FUNCTION_BLOCK SifbManagementControls
  (* Standard: 61499-2 *)
  (* Version 0.1, 2019-00-29, hpea485, UOA *)
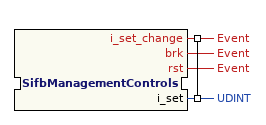
  EVENT_OUTPUT
    i_set_change WITH i_set;
    brk;
    rst;
  END_EVENT
  VAR_OUTPUT
    i_set : UDINT;
  END_VAR
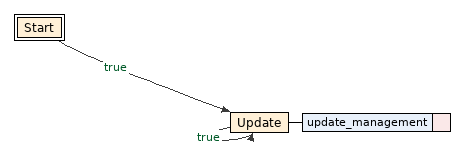
  EC_STATES
    Start;
    Update : update_management;
  END_STATES
  EC_TRANSITIONS
    Start TO Update := true;
    Update TO Update := true;
  END_TRANSITIONS
  ALGORITHM update_management IN C:
int sw_break = ((SWITCHES & 0b0001) != 0);
int sw_reset = ((SWITCHES & 0b0010) != 0);
int sw_iseth = ((SWITCHES & 0b0100) != 0);

if(sw_iseth == 1 && (int)(me->i_set) != 100) {
	//switch is pressed
	me->i_set = 1000.0;
	me->outputEvents.event.i_set_change = 1;
}
if(sw_iseth == 0 && (int)(me->i_set) != 10) {
	//switch is pressed
	me->i_set = 10.0;
	me->outputEvents.event.i_set_change = 1;
}
me->outputEvents.event.brk = (sw_break > 0);
me->outputEvents.event.rst = (sw_reset > 0);
  END_ALGORITHM
END_FUNCTION_BLOCK
